// TIA Portal V18 export
DATA_BLOCK "OP10_GeneralAnalogDB"   // DB1080
{ S7_Optimized_Access := 'TRUE' }
// stored: AutoNumber false, MemoryReserve 0
   VAR RETAIN
      aDev : Array[1..2] of "ST_GeneralAnalog";
   END_VAR
BEGIN
END_DATA_BLOCK
